// TwinCAT 3 PLC project PlcTemplate
// Title: PlcTemplate
// Company: Vortex.Library
// ProjectVersion: 0.6.0.913
// ProgramVersion: 3.1.4023.0
// libraries:
//   Tc2_Standard, * (Beckhoff Automation GmbH)
//   Tc2_System, * (Beckhoff Automation GmbH)
//   Tc3_Module, * (Beckhoff Automation GmbH)
//   TcoCore, 0.6.0.913 (Vortex.Library)
// project tree:
//   / PlcTask.TcTTO (not stored)
//   POUs/ MAIN.TcPOU, SampleContext.TcPOU
//   POUs/SampleComponent/ SampleComponent.TcPOU, SampleTaskFunctionBuffer.TcDUT, SampleTaskIteration.TcPOU
// real-time tasks:
//   TASK PlcTask: cycle T#10ms, priority 20, ADS port 350
//   TASK PlcTask1: cycle T#10ms, priority 21, ADS port 351

// ---- POUs/SampleComponent/SampleTaskFunctionBuffer.TcDUT
TYPE SampleTaskFunctionBuffer :
STRUCT
    x : LREAL;
    y : LREAL;
END_STRUCT
END_TYPE

// ---- POUs/MAIN.TcPOU
PROGRAM MAIN
VAR
    _sampleContext : SampleContext;
END_VAR

_sampleContext.Run();

END_PROGRAM

// ---- POUs/SampleContext.TcPOU
FUNCTION_BLOCK SampleContext EXTENDS TcoCore.TcoContext
VAR
    _sampleComponent : SampleComponent(THIS^);
END_VAR

(*~
    <docu>
        <summary>
            Main method of the TcoContext. This is the entry point of any control logic that belongs to this context.
            The call of this method is ensured by calling the <c>InstanceName.Run()</c> method, and it must not be called explicitly.
            This method is abstract, and it must be overridden in derived block.
        </summary>
    </docu>
~*)
METHOD PROTECTED Main
_sampleComponent.Service();
_sampleComponent();
END_METHOD

END_FUNCTION_BLOCK

// ---- POUs/SampleComponent/SampleComponent.TcPOU
(*~
    <docu>
        <summary>Sample component for inspiration</summary>
    </docu>
~*)
FUNCTION_BLOCK SampleComponent EXTENDS TcoCore.TcoComponent
VAR
    (*~
        <docu>
            <summary>Counter</summary>
            <remarks>
                > [!IMPORTANT]
                > This member is ignored when rendering.
            </remarks>
        </docu>
    ~*)
    {attribute clr [RenderIgnore()]}
    _counter : INT;
END_VAR
VAR
    (*~
        <docu>
            <summary>Counter</summary>
            <remarks>
                > [!IMPORTANT]
                > This member is readonly.
            </remarks>
        </docu>
    ~*)
    {attribute addProperty Name "Add Result"}
    {attribute clr [ReadOnly()]}
    _addResult : INT;
    {attribute addProperty Name "A"}
    _addNumberOne : INT;
    {attribute addProperty Name "B"}
    _addNumberTwo : INT;
END_VAR
VAR
    _sampleTask : SampleTaskIteration(THIS^);
END_VAR

_addResult := THIS^.AddTwoNumbers(_addNumberOne, _addNumberTwo);
_sampleTask();

(*~
    <docu>
        <summary>Adds two numbers</summary>
        <returns>Sum of two numbers</returns>
    </docu>
~*)
METHOD AddTwoNumbers : INT
VAR_INPUT
    NumberOne : INT;
    NumberTwo : INT;
END_VAR
AddTwoNumbers := NumberOne + NumberTwo;
END_METHOD

{attribute 'TcRpcEnable'}
METHOD INTERNAL AddTwoNumbersTest : INT
VAR_INPUT
    NumberOne : INT;
    NumberTwo : INT;
END_VAR
AddTwoNumbersTest := THIS^.AddTwoNumbers(NumberOne, NumberTwo);
END_METHOD

METHOD FB_init : BOOL
VAR_INPUT
    bInitRetains : BOOL; // if TRUE, the retain variables are initialized (warm start / cold start)
    bInCopyCode : BOOL; // if TRUE, the instance afterwards gets moved into the copy code (online change)
    ParentObject : ITcoObject;
END_VAR
END_METHOD

(*~
    <docu>
        <summary>
            Restores this instance to the Ready state. Can be called explicitly or from within one of the restore mechanisms.
        </summary>
    </docu>
~*)
METHOD Restore : ITcoRestorable
END_METHOD

(*~
    <docu>
        <summary>
            Custom service (manual, maintenance) logic.
            This method must be implemented in derived class.
        </summary>
    </docu>
~*)
METHOD PROTECTED ServiceMode
END_METHOD

METHOD WaitForModulo : BOOL
VAR_INPUT
    Modulo : INT;
END_VAR
_counter := _counter + 1;
WaitForModulo := _counter MOD Modulo = 0;
END_METHOD

{attribute 'TcRpcEnable'}
METHOD INTERNAL WaitForModuloTest : BOOL
VAR_INPUT
    Modulo : INT;
END_VAR
WaitForModuloTest := THIS^.WaitForModulo(Modulo);
END_METHOD

END_FUNCTION_BLOCK

// ---- POUs/SampleComponent/SampleTaskIteration.TcPOU
FUNCTION_BLOCK SampleTaskIteration EXTENDS TcoCore.TcoTask
VAR
    _x : LREAL;
    _y : LREAL;
    _d : LREAL;
    {attribute addProperty Minimum 100}
    {attribute addProperty Maximum 1000}
    _iterations : INT;
    _currentIteration : INT;
END_VAR

IF (Execute()) THEN
    _y := SIN(_x);
    _x := _x + _d;
    _currentIteration := _currentIteration + 1;
    DoneWhen(_currentIteration >= _iterations);
END_IF

METHOD FB_init : BOOL
VAR_INPUT
    bInitRetains : BOOL; // if TRUE, the retain variables are initialized (warm start / cold start)
    bInCopyCode : BOOL; // if TRUE, the instance afterwards gets moved into the copy code (online change)
    ParentObject : ITcoObject;
END_VAR
END_METHOD

(*~
    <docu>
        <summary>
            Restores this instance to the Ready state. Can be called explicitly or from within one of the restore mechanisms.
            <para>
                See also <see cref="PlcDocu.TcoCore.TcoTask.AutoRestorable()"/>
            </para>
        </summary>
    </docu>
~*)
METHOD Restore : ITcoRestorable
SUPER^.Restore();
_x := 0.0;
_y := 0.0;
_currentIteration := 0;
END_METHOD

END_FUNCTION_BLOCK
